PROGRAM Robot
VAR
	// Goto Home
	ABBGotoHome_Control: ABBGotoHome;
	GotoHome: BOOL;
	GotoHomeDone: BOOL;
	
	// Go to AGV
	ABBGotoAGVPosByScanner_Control: ABBGotoAGVPos;
	GotoAGVByScanner: BOOL;
	GotoAGVByScannerDone: BOOL;
	
	// Go to AGV
	ABBGotoAGVPosByAssembly_Control: ABBGotoAGVPos;
	GotoAGVByAssembly: BOOL;
	GotoAGVByAssemblyDone: BOOL;
	
	// Go to Scanner
	ABBGotoScannerFromAGV_Control: ABBGotoScanner;
	ABBGotoScannerFromBuffer_Control: ABBGotoScanner;
	GotoScannerFromBuffer: BOOL;
	GotoScannerFromAGV: BOOL;
	GotoScannerFromBufferDone: BOOL;
	GotoScannerFromAGVDone: BOOL;
	
	// Go to Table
	ABBGotoTableByAGV_Control: ABBGotoTable;
	GotoTableByAGV: BOOL;
	GotoTableByAGVDone: BOOL;
	
	ABBGotoTableByScanner_Control: ABBGotoTable;
	GotoTableByScanner: BOOL;
	GotoTableDoneByScanner: BOOL;
	
	ABBGotoTableByAssembly_Control: ABBGotoTable;
	GotoTableByAssembly: BOOL;
	GotoTableDoneByAssembly: BOOL;
	
	// Go to Buffer
	ABBGotoBuffer_Control: ABBGotoBuffer;
	GotoBuffer: BOOL;
	GotoBufferDone: BOOL;
	
	// PickLeave Container AGV
	ABBPickLeaveContainerAGV_Control: ABBPickLeaveContainerAGV;
	PickAGV: BOOL;
	LeaveAGV: BOOL;
	PickLeaveAGVDone: BOOL;
	
	// PickLeave Scanner
	ABBPickLeaveScannerFromBuffer_Control: ABBPickLeaveScanner;
	ABBPickLeaveScannerFromAGV_Control: ABBPickLeaveScanner;
	PickScannerFromBuffer: BOOL;
	LeaveScannerFromBuffer: BOOL;
	PickLeaveScannerFromBufferDone: BOOL;
	PickScannerFromAGV: BOOL;
	LeaveScannerFromAGV: BOOL;
	PickLeaveScannerFromAGVDone: BOOL;
	
	
	// PickLeave Buffer
	ABBPickLeaveBuffer_Control: ABBPickLeaveBuffer;
	PickBuffer: BOOL;
	LeaveBuffer: BOOL;
	PickLeaveBufferDone: BOOL;
	
	// PickLeave Table
	ABBPickLeaveTable_Control: ABBPickLeaveContaineronTable;
	PickTable: BOOL;
	LeaveTable: BOOL;
	PickLeaveTableDone: BOOL;
	
	// Scan parts
	ABBScanContainer_Control: ABBScanContainer;
	ScanContainer: BOOL;
	ScanContainerPartAvailable: BOOL;
	ScanContainerDone: BOOL;
	
	// Assemble parts
	ABBAssemble_Control: ABBAssemble;
	Assemble: BOOL;
	AssembleBufferId: INT;
	AssemblePartId: INT;
	AssembleDone: BOOL;
	
	// Read sensor
	ABBScannerStationByBuffer_Control: ABBScannerStation;
	ABBScannerStationByAGV_Control: ABBScannerStation;
	ReadSensorByBuffer: BOOL;
	ReadSensorByAGV: BOOL;
	ReadSensorByBufferDone: BOOL;
	ReadSensorByAGVDone: BOOL;
	
	
	// Read sensor
	IdentifyPartFB: IdentifyPart;
	IdentifyPart_Control: IdentifyPart;
	ScanPartId: INT;
END_VAR

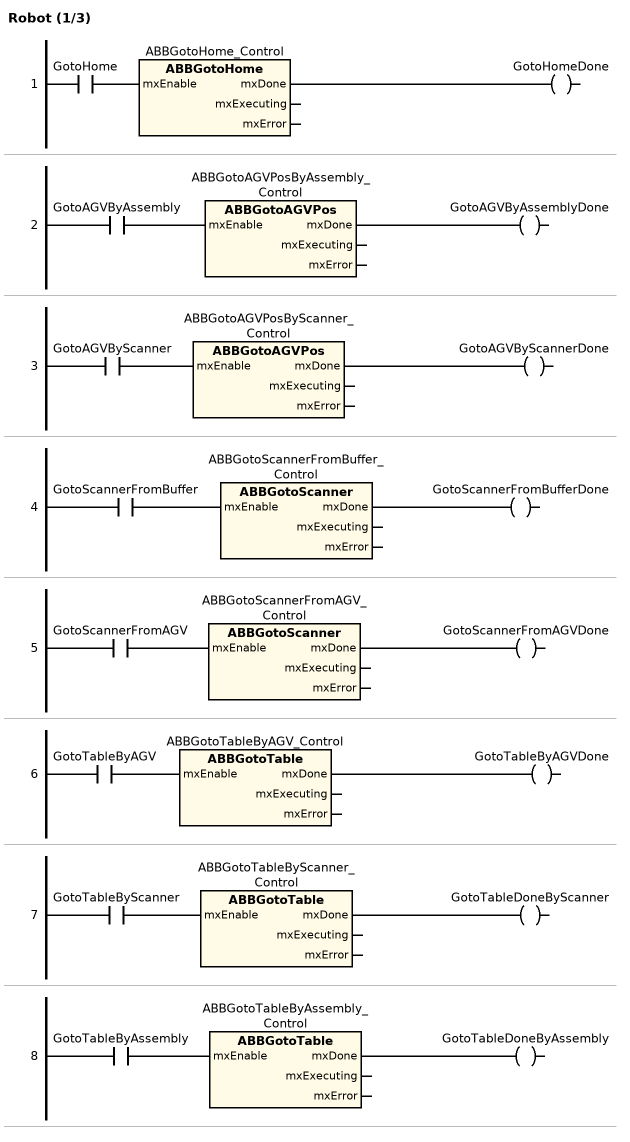
// NETWORK 1
ABBGotoHome_Control(mxEnable := GotoHome); // ABBGotoHome
GotoHomeDone := ABBGotoHome_Control.mxDone;

// NETWORK 2
ABBGotoAGVPosByAssembly_Control(mxEnable := GotoAGVByAssembly); // ABBGotoAGVPos
GotoAGVByAssemblyDone := ABBGotoAGVPosByAssembly_Control.mxDone;

// NETWORK 3
ABBGotoAGVPosByScanner_Control(mxEnable := GotoAGVByScanner); // ABBGotoAGVPos
GotoAGVByScannerDone := ABBGotoAGVPosByScanner_Control.mxDone;

// NETWORK 4
ABBGotoScannerFromBuffer_Control(mxEnable := GotoScannerFromBuffer); // ABBGotoScanner
GotoScannerFromBufferDone := ABBGotoScannerFromBuffer_Control.mxDone;

// NETWORK 5
ABBGotoScannerFromAGV_Control(mxEnable := GotoScannerFromAGV); // ABBGotoScanner
GotoScannerFromAGVDone := ABBGotoScannerFromAGV_Control.mxDone;

// NETWORK 6
ABBGotoTableByAGV_Control(mxEnable := GotoTableByAGV); // ABBGotoTable
GotoTableByAGVDone := ABBGotoTableByAGV_Control.mxDone;

// NETWORK 7
ABBGotoTableByScanner_Control(mxEnable := GotoTableByScanner); // ABBGotoTable
GotoTableDoneByScanner := ABBGotoTableByScanner_Control.mxDone;

// NETWORK 8
ABBGotoTableByAssembly_Control(mxEnable := GotoTableByAssembly); // ABBGotoTable
GotoTableDoneByAssembly := ABBGotoTableByAssembly_Control.mxDone;

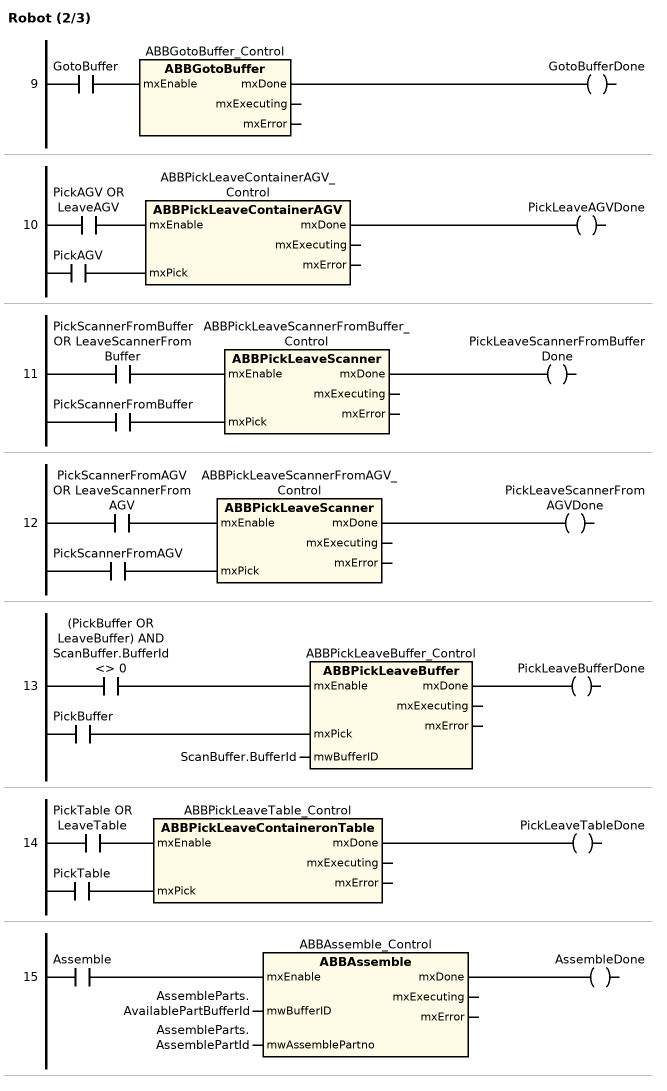
// NETWORK 9
ABBGotoBuffer_Control(mxEnable := GotoBuffer); // ABBGotoBuffer
GotoBufferDone := ABBGotoBuffer_Control.mxDone;

// NETWORK 10
ABBPickLeaveContainerAGV_Control(mxEnable := PickAGV OR LeaveAGV, mxPick := PickAGV); // ABBPickLeaveContainerAGV
PickLeaveAGVDone := ABBPickLeaveContainerAGV_Control.mxDone;

// NETWORK 11
ABBPickLeaveScannerFromBuffer_Control(mxEnable := PickScannerFromBuffer OR LeaveScannerFromBuffer, mxPick := PickScannerFromBuffer); // ABBPickLeaveScanner
PickLeaveScannerFromBufferDone := ABBPickLeaveScannerFromBuffer_Control.mxDone;

// NETWORK 12
ABBPickLeaveScannerFromAGV_Control(mxEnable := PickScannerFromAGV OR LeaveScannerFromAGV, mxPick := PickScannerFromAGV); // ABBPickLeaveScanner
PickLeaveScannerFromAGVDone := ABBPickLeaveScannerFromAGV_Control.mxDone;

// NETWORK 13
ABBPickLeaveBuffer_Control(
    mxEnable := (PickBuffer OR LeaveBuffer) AND ScanBuffer.BufferId <> 0,
    mxPick := PickBuffer,
    mwBufferID := ScanBuffer.BufferId); // ABBPickLeaveBuffer
PickLeaveBufferDone := ABBPickLeaveBuffer_Control.mxDone;

// NETWORK 14
ABBPickLeaveTable_Control(mxEnable := PickTable OR LeaveTable, mxPick := PickTable); // ABBPickLeaveContaineronTable
PickLeaveTableDone := ABBPickLeaveTable_Control.mxDone;

// NETWORK 15
ABBAssemble_Control(
    mxEnable := Assemble,
    mwBufferID := AssembleParts.AvailablePartBufferId,
    mwAssemblePartno := AssembleParts.AssemblePartId); // ABBAssemble
AssembleDone := ABBAssemble_Control.mxDone;

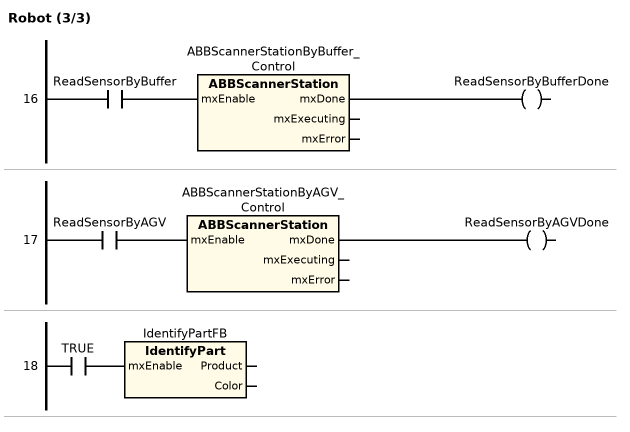
// NETWORK 16
ABBScannerStationByBuffer_Control(mxEnable := ReadSensorByBuffer); // ABBScannerStation
ReadSensorByBufferDone := ABBScannerStationByBuffer_Control.mxDone;

// NETWORK 17
ABBScannerStationByAGV_Control(mxEnable := ReadSensorByAGV); // ABBScannerStation
ReadSensorByAGVDone := ABBScannerStationByAGV_Control.mxDone;

// NETWORK 18
IdentifyPartFB(mxEnable := TRUE); // IdentifyPart

END_PROGRAM

(* stored: Version 1.1.0.1, ProductVersion 3.1.4024.12
   POU Robot: Id {542b48bc-9240-4d89-91b4-f34cda73c2e6}, SpecialFunc None *)
